(* PLC project AufgSer3, Beckhoff Automation GmbH TwinCAT PLC Control 3.5.13.21 *)
(* stored: creationDateTime 2022-04-25T13:35:18.1005355, modificationDateTime 2022-04-25T13:35:18.105542 *)

FUNCTION F_Sine : REAL
VAR_INPUT
	A		: REAL;	// Amplitude
	yoff	: REAL; // offset
	w		: REAL; // Kreisfrequenz (rad/s)
	t		: REAL; // Time (s)
END_VAR
VAR
END_VAR

            F_Sine := (A * SIN(w*t)) + yoff;
          
END_FUNCTION
